{attribute 'GeneratedUsingTerminal: EL2596-0000-0017'}
{attribute addProperty BoxType "EL2596-0000-0017"}
{attribute addProperty Id "EtcSlaveTerminalBaseDOX_StatusAT %I*DOX_Status_F52B34D37DOX_ControlAT %Q*DOX_Control_B191BB935WcStateAT %I*WcState_9091E0EB2InfoDataAT %I*InfoData_32EB74EA10"}
{attribute addProperty CRC "245164624"}
{attribute addProperty Size "24"}
TYPE EL2596_0E9CEA50 EXTENDS EtcSlaveTerminalBase :
STRUCT
	{attribute addProperty Name "DOX_Status"}
	DOX_Status : DOX_Status_F52B34D3;
	{attribute addProperty Name "DOX_Control"}
	DOX_Control : DOX_Control_B191BB93;
	{attribute addProperty Name "WcState"}
	WcState : WcState_9091E0EB;
	{attribute addProperty Name "InfoData"}
	InfoData : InfoData_32EB74EA;
END_STRUCT
END_TYPE

(* stored: Version 1.2.0.0, ProductVersion 3.1.4024.9
   DUT EL2596_0E9CEA50: Id {c4de0a2a-4ffb-4434-a07b-0906d2ce1cd1} *)
